{attribute 'qualified_only'}
VAR_GLOBAL
	monitoredValues : ARRAY[0..16] OF MonitoredValue;
END_VAR

(* stored: Version 1.1.0.1, ProductVersion 3.1.4024.12
   GVL gScaledIO: Id {d4b685b7-b49f-4044-b0e2-abfab7a9f699} *)
